(* Logix 5000 project; controller L62 1756-L62 rev 20.19; software revision 20.05 *)

TASK MainTask (continuous, watchdog 500 ms) : MainProgram

MODULES
   Local : 1756-L62 (ICP 2, rev 20.19)
END_MODULES

VAR_GLOBAL   (* controller tags *)
   InstanciaMSG : MESSAGE;
        MessageParameters(ServiceCode := 16#0f68, LocalElement := Serial_data_control[0], ...)
   Serial_data_control : INT[10] := ([0] := 10, [1] := 2, [2] := 3, [3] := 4, [4] := 4, [5] := 4, [6] := 5, [7] := 6, [8] := 7, [9] := 8);
END_VAR

PROGRAM MainProgram   (* main routine MainRoutine *)
VAR
   Trigger : BOOL := 1;
END_VAR

ROUTINE MainRoutine   (* ladder *)
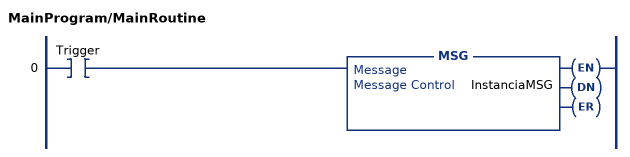
   0: XIC(Trigger)MSG(InstanciaMSG);
END_ROUTINE
END_PROGRAM
